// TIA Portal V17 export
// export: Created 2023-12-22T15:05:26.1388386Z, ExportSetting WithDefaults, DisplayName Totally Integrated Automation Portal, DisplayVersion V17, DisplayName TIA Portal Openness, DisplayVersion V17, DisplayName TIA Portal Version Control Interface, DisplayVersion V17, DisplayName STEP 7 Professional, DisplayVersion V17, DisplayName STEP 7 Safety, DisplayVersion V17, DisplayName WinCC Advanced, DisplayVersion V17
FUNCTION "Comm_Scada_FC" : Void   // FC1, LAD
{ S7_Optimized_Access := 'TRUE' }
VERSION : 0.1
// stored: AutoNumber true, IsIECCheckEnabled false, SetENOAutomatically false, UDAEnableTagReadback false
BEGIN

REGION Network 1: Output Запуски
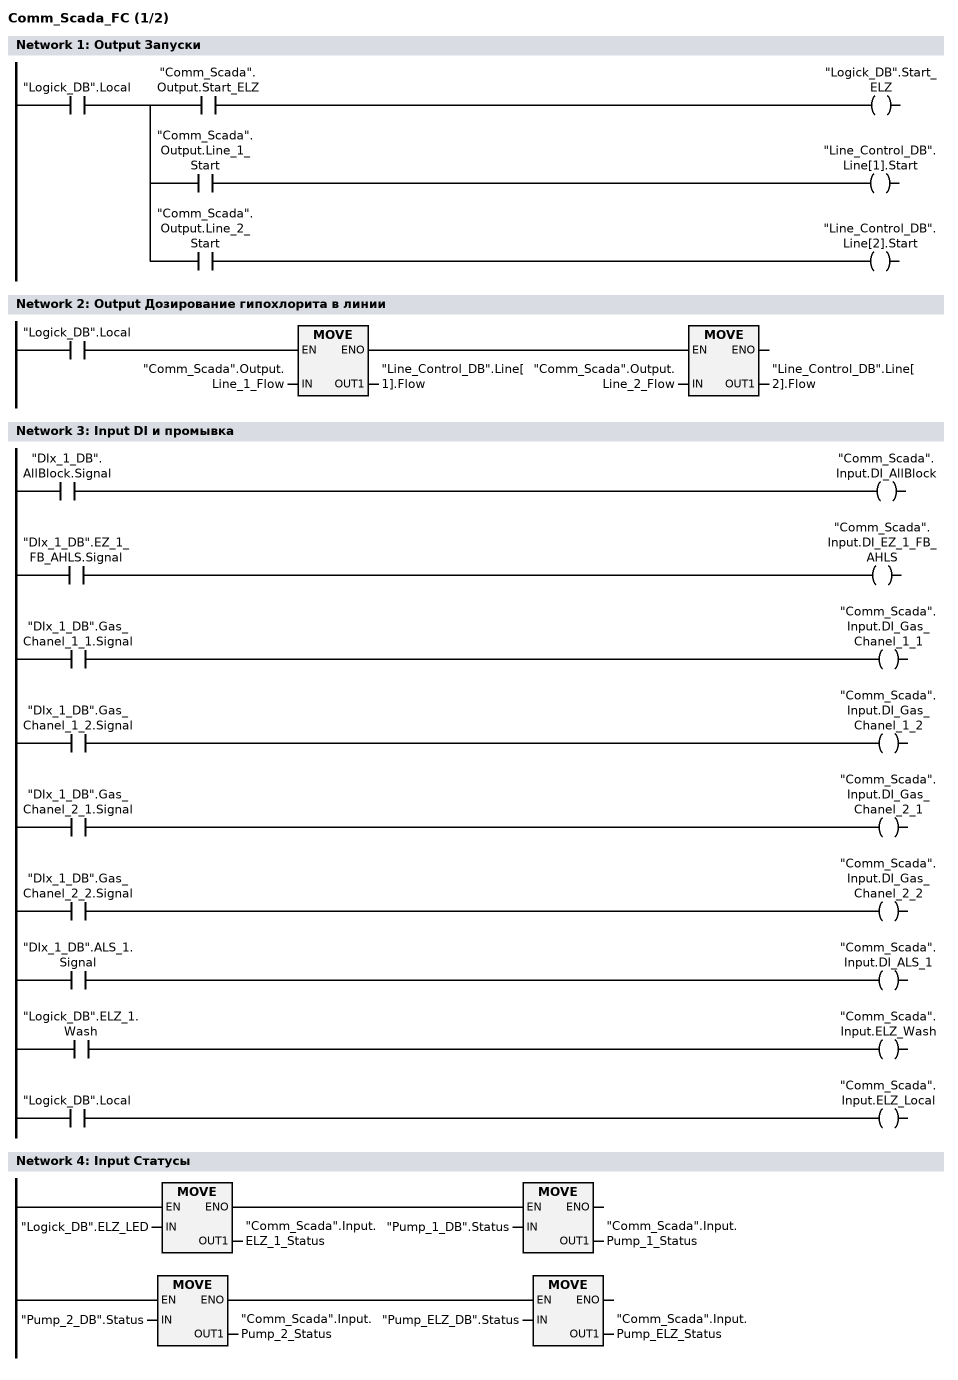
   RUNG wire#powerrail
      Contact( "Logick_DB".Local )
      wire#w1
      Contact( "Comm_Scada".Output.Start_ELZ )
      Coil( "Logick_DB".Start_ELZ )
   END_RUNG
   RUNG wire#w1
      Contact( "Comm_Scada".Output.Line_1_Start )
      Coil( "Line_Control_DB".Line[1].Start )
   END_RUNG
   RUNG wire#w1
      Contact( "Comm_Scada".Output.Line_2_Start )
      Coil( "Line_Control_DB".Line[2].Start )
   END_RUNG
   // the same network as SCL:
   "Logick_DB".Start_ELZ := "Logick_DB".Local AND "Comm_Scada".Output.Start_ELZ;
   "Line_Control_DB".Line[1].Start := "Logick_DB".Local AND "Comm_Scada".Output.Line_1_Start;
   "Line_Control_DB".Line[2].Start := "Logick_DB".Local AND "Comm_Scada".Output.Line_2_Start;
END_REGION

REGION Network 2: Output Дозирование гипохлорита в линии
   RUNG wire#powerrail
      Contact( "Logick_DB".Local )
      Move(in := "Comm_Scada".Output.Line_1_Flow, out1 => "Line_Control_DB".Line[1].Flow)
      Move(in := "Comm_Scada".Output.Line_2_Flow, out1 => "Line_Control_DB".Line[2].Flow)
   END_RUNG
   // the same network as SCL:
   IF "Logick_DB".Local THEN
       "Line_Control_DB".Line[1].Flow := "Comm_Scada".Output.Line_1_Flow;
       "Line_Control_DB".Line[2].Flow := "Comm_Scada".Output.Line_2_Flow;
   END_IF;
END_REGION

REGION Network 3: Input DI и промывка
   RUNG wire#powerrail
      Contact( "DIx_1_DB".AllBlock.Signal )
      Coil( "Comm_Scada".Input.DI_AllBlock )
   END_RUNG
   RUNG wire#powerrail
      Contact( "DIx_1_DB".EZ_1_FB_AHLS.Signal )
      Coil( "Comm_Scada".Input.DI_EZ_1_FB_AHLS )
   END_RUNG
   RUNG wire#powerrail
      Contact( "DIx_1_DB".Gas_Chanel_1_1.Signal )
      Coil( "Comm_Scada".Input.DI_Gas_Chanel_1_1 )
   END_RUNG
   RUNG wire#powerrail
      Contact( "DIx_1_DB".Gas_Chanel_1_2.Signal )
      Coil( "Comm_Scada".Input.DI_Gas_Chanel_1_2 )
   END_RUNG
   RUNG wire#powerrail
      Contact( "DIx_1_DB".Gas_Chanel_2_1.Signal )
      Coil( "Comm_Scada".Input.DI_Gas_Chanel_2_1 )
   END_RUNG
   RUNG wire#powerrail
      Contact( "DIx_1_DB".Gas_Chanel_2_2.Signal )
      Coil( "Comm_Scada".Input.DI_Gas_Chanel_2_2 )
   END_RUNG
   RUNG wire#powerrail
      Contact( "DIx_1_DB".ALS_1.Signal )
      Coil( "Comm_Scada".Input.DI_ALS_1 )
   END_RUNG
   RUNG wire#powerrail
      Contact( "Logick_DB".ELZ_1.Wash )
      Coil( "Comm_Scada".Input.ELZ_Wash )
   END_RUNG
   RUNG wire#powerrail
      Contact( "Logick_DB".Local )
      Coil( "Comm_Scada".Input.ELZ_Local )
   END_RUNG
   // the same network as SCL:
   "Comm_Scada".Input.DI_AllBlock := "DIx_1_DB".AllBlock.Signal;
   "Comm_Scada".Input.DI_EZ_1_FB_AHLS := "DIx_1_DB".EZ_1_FB_AHLS.Signal;
   "Comm_Scada".Input.DI_Gas_Chanel_1_1 := "DIx_1_DB".Gas_Chanel_1_1.Signal;
   "Comm_Scada".Input.DI_Gas_Chanel_1_2 := "DIx_1_DB".Gas_Chanel_1_2.Signal;
   "Comm_Scada".Input.DI_Gas_Chanel_2_1 := "DIx_1_DB".Gas_Chanel_2_1.Signal;
   "Comm_Scada".Input.DI_Gas_Chanel_2_2 := "DIx_1_DB".Gas_Chanel_2_2.Signal;
   "Comm_Scada".Input.DI_ALS_1 := "DIx_1_DB".ALS_1.Signal;
   "Comm_Scada".Input.ELZ_Wash := "Logick_DB".ELZ_1.Wash;
   "Comm_Scada".Input.ELZ_Local := "Logick_DB".Local;
END_REGION

REGION Network 4: Input Статусы
   RUNG wire#powerrail
      Move(in := "Logick_DB".ELZ_LED, out1 => "Comm_Scada".Input.ELZ_1_Status)
      Move(in := "Pump_1_DB".Status, out1 => "Comm_Scada".Input.Pump_1_Status)
   END_RUNG
   RUNG wire#powerrail
      Move(in := "Pump_2_DB".Status, out1 => "Comm_Scada".Input.Pump_2_Status)
      Move(in := "Pump_ELZ_DB".Status, out1 => "Comm_Scada".Input.Pump_ELZ_Status)
   END_RUNG
   // the same network as SCL:
   "Comm_Scada".Input.ELZ_1_Status := "Logick_DB".ELZ_LED;
   "Comm_Scada".Input.Pump_1_Status := "Pump_1_DB".Status;
   "Comm_Scada".Input.Pump_2_Status := "Pump_2_DB".Status;
   "Comm_Scada".Input.Pump_ELZ_Status := "Pump_ELZ_DB".Status;
END_REGION

REGION Network 5: Input Дозирование гипохлорита
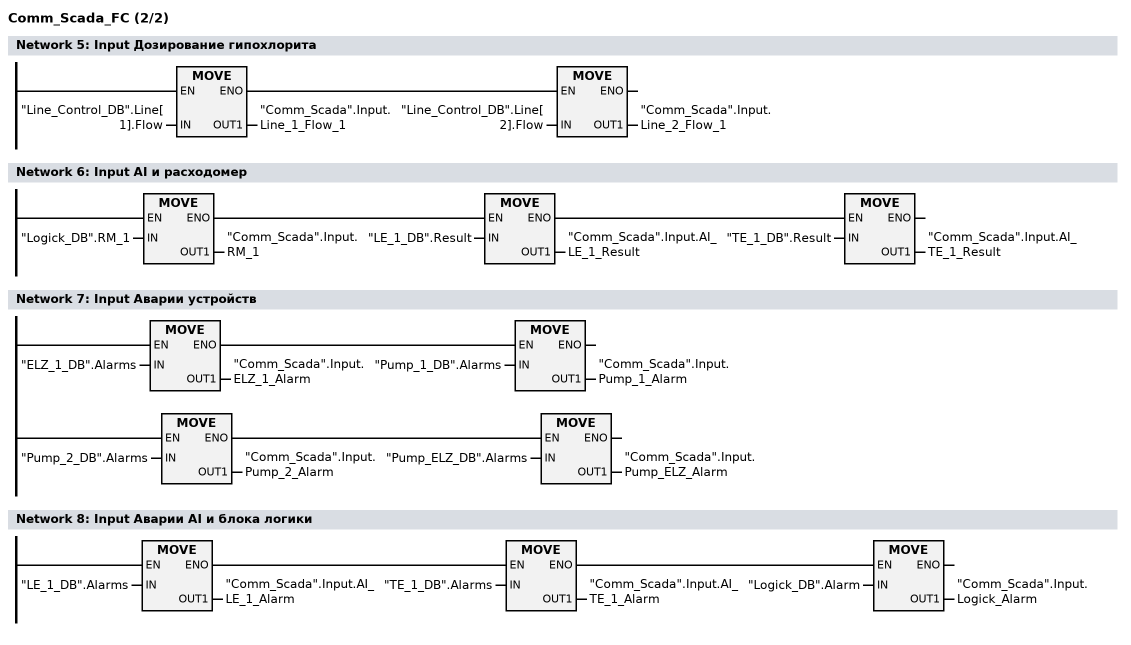
   RUNG wire#powerrail
      Move(in := "Line_Control_DB".Line[1].Flow, out1 => "Comm_Scada".Input.Line_1_Flow_1)
      Move(in := "Line_Control_DB".Line[2].Flow, out1 => "Comm_Scada".Input.Line_2_Flow_1)
   END_RUNG
   // the same network as SCL:
   "Comm_Scada".Input.Line_1_Flow_1 := "Line_Control_DB".Line[1].Flow;
   "Comm_Scada".Input.Line_2_Flow_1 := "Line_Control_DB".Line[2].Flow;
END_REGION

REGION Network 6: Input AI и расходомер
   RUNG wire#powerrail
      Move(in := "Logick_DB".RM_1, out1 => "Comm_Scada".Input.RM_1)
      Move(in := "LE_1_DB".Result, out1 => "Comm_Scada".Input.AI_LE_1_Result)
      Move(in := "TE_1_DB".Result, out1 => "Comm_Scada".Input.AI_TE_1_Result)
   END_RUNG
   // the same network as SCL:
   "Comm_Scada".Input.RM_1 := "Logick_DB".RM_1;
   "Comm_Scada".Input.AI_LE_1_Result := "LE_1_DB".Result;
   "Comm_Scada".Input.AI_TE_1_Result := "TE_1_DB".Result;
END_REGION

REGION Network 7: Input Аварии устройств
   RUNG wire#powerrail
      Move(in := "ELZ_1_DB".Alarms, out1 => "Comm_Scada".Input.ELZ_1_Alarm)
      Move(in := "Pump_1_DB".Alarms, out1 => "Comm_Scada".Input.Pump_1_Alarm)
   END_RUNG
   RUNG wire#powerrail
      Move(in := "Pump_2_DB".Alarms, out1 => "Comm_Scada".Input.Pump_2_Alarm)
      Move(in := "Pump_ELZ_DB".Alarms, out1 => "Comm_Scada".Input.Pump_ELZ_Alarm)
   END_RUNG
   // the same network as SCL:
   "Comm_Scada".Input.ELZ_1_Alarm := "ELZ_1_DB".Alarms;
   "Comm_Scada".Input.Pump_1_Alarm := "Pump_1_DB".Alarms;
   "Comm_Scada".Input.Pump_2_Alarm := "Pump_2_DB".Alarms;
   "Comm_Scada".Input.Pump_ELZ_Alarm := "Pump_ELZ_DB".Alarms;
END_REGION

REGION Network 8: Input Аварии AI и блока логики
   RUNG wire#powerrail
      Move(in := "LE_1_DB".Alarms, out1 => "Comm_Scada".Input.AI_LE_1_Alarm)
      Move(in := "TE_1_DB".Alarms, out1 => "Comm_Scada".Input.AI_TE_1_Alarm)
      Move(in := "Logick_DB".Alarm, out1 => "Comm_Scada".Input.Logick_Alarm)
   END_RUNG
   // the same network as SCL:
   "Comm_Scada".Input.AI_LE_1_Alarm := "LE_1_DB".Alarms;
   "Comm_Scada".Input.AI_TE_1_Alarm := "TE_1_DB".Alarms;
   "Comm_Scada".Input.Logick_Alarm := "Logick_DB".Alarm;
END_REGION
END_FUNCTION
